(* CoDeSys 2.3 export: EV_SIMPLE.EXP *)

(* Data type *)
TYPE EV_Simple :
STRUCT
	Activa : BOOL;
END_STRUCT
END_TYPE
